PROGRAM MAIN
VAR
END_VAR

END_PROGRAM

(* stored: Version 1.1.0.1
   POU MAIN: Id {6b8117ec-acc4-4b54-80de-cfad493a19f8} *)
